Fanuc KAREL source: compact_preamble.KL

PROGRAM KB00103
%NOLOCKGROUP
VAR
P1:INTEGER;P2:INTEGER;P3 : STRING[80];P4:INTEGER;P5:INTEGER;P6:INTEGER;P7:INTEGER;P8:INTEGER;P9:INTEGER;P10 : ARRAY[4] OF STRING[80];P11:INTEGER
BEGIN
P1=1
P2=1
P3='A'
P4=1
P5=1
P6=1
P7=1
P8=1
P9=1
P11=1
INI_DYN_DISP(P1,P2,P3,P4,P5,P6,P7,P8,P9,P10,P11)
END KB00103
